% RSLogix 500 project P7 - Sensor Calibration.RSS, saved by version 8.30.00.16 %
PROJECT "P7"    % processor: Bul.1763 MicroLogix 1100 Series B %

PROGRAM FILES
  LAD 2 "MAIN"  3 rungs
  LAD 3 "IO"  3 rungs
  LAD 4 "SAMPLING"  4 rungs
  LAD 5 "CALIBRATE"  11 rungs

DATA FILES
  O0 OUTPUT  4 elements
  I1 INPUT  6 elements
  S2 STATUS  66 elements
  B3 BINARY  1 elements
  T4 TIMER  3 elements
  C5 COUNTER  1 elements
  R6 CONTROL  1 elements
  N7 INTEGER  8 elements
  F8 FLOAT  5 elements
  PD9 PD  1 elements

LADDER 2 "MAIN"
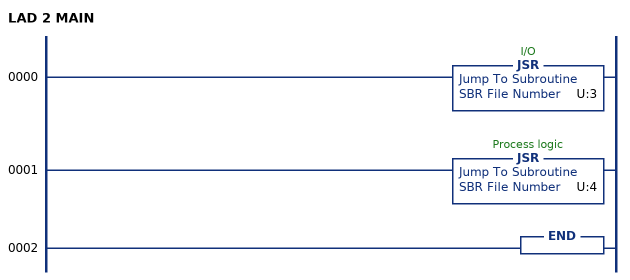
% Rung: 0 %
SOR JSR U:3 EOR
%   U:3  "I/O" %
% Rung: 1 %
SOR JSR U:4 EOR
%   U:4  "Process logic" %
% Rung: 2 %
SOR END EOR

LADDER 3 "IO"
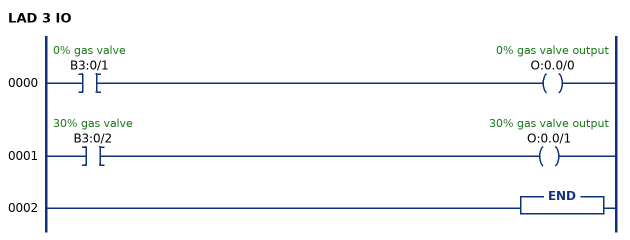
% Rung: 0 %
SOR XIC B3:0/1 OTE O:0.0/0 EOR
%   B3:0/1  "0% gas valve" %
%   O:0.0/0  "0% gas valve output" %
% Rung: 1 %
SOR XIC B3:0/2 OTE O:0.0/1 EOR
%   B3:0/2  "30% gas valve" %
%   O:0.0/1  "30% gas valve output" %
% Rung: 2 %
SOR END EOR

LADDER 4 "SAMPLING"
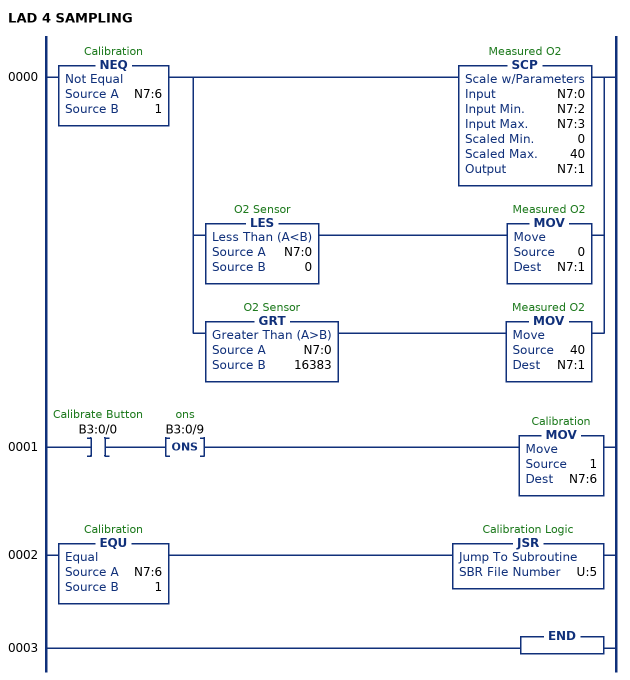
% Rung: 0 %
SOR NEQ N7:6 1 BST SCP N7:0 N7:2 N7:3 0 40 N7:1 NXB LES N7:0 0 MOV 0 N7:1 NXB GRT N7:0 16383 MOV 40 N7:1 BND EOR
%   N7:6  "Calibration" %
%   N7:0  "O2 Sensor" %
%   N7:2  "O2 min" %
%   N7:3  "O2 max" %
%   N7:1  "Measured O2" %
% Rung: 1 %
SOR XIC B3:0/0 ONS B3:0/9 MOV 1 N7:6 EOR
%   B3:0/0  "Calibrate Button" %
%   B3:0/9  "ons" %
%   N7:6  "Calibration" %
% Rung: 2 %
SOR EQU N7:6 1 JSR U:5 EOR
%   N7:6  "Calibration" %
%   U:5  "Calibration Logic" %
% Rung: 3 %
SOR END EOR

LADDER 5 "CALIBRATE"
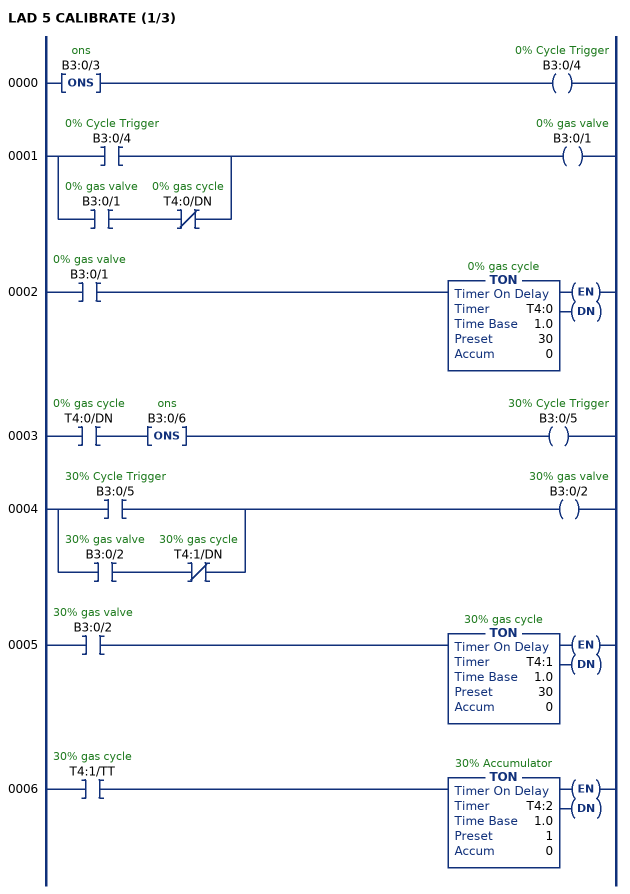
% Rung: 0 %
SOR ONS B3:0/3 OTE B3:0/4 EOR
%   B3:0/3  "ons" %
%   B3:0/4  "0% Cycle Trigger" %
% Rung: 1 %
SOR BST XIC B3:0/4 NXB XIC B3:0/1 XIO T4:0/DN BND OTE B3:0/1 EOR
%   B3:0/4  "0% Cycle Trigger" %
%   B3:0/1  "0% gas valve" %
%   T4:0  "0% gas cycle" %
% Rung: 2 %
SOR XIC B3:0/1 TON T4:0 1.0 30 0 EOR
%   B3:0/1  "0% gas valve" %
%   T4:0  "0% gas cycle" %
% Rung: 3 %
SOR XIC T4:0/DN ONS B3:0/6 OTE B3:0/5 EOR
%   T4:0  "0% gas cycle" %
%   B3:0/6  "ons" %
%   B3:0/5  "30% Cycle Trigger" %
% Rung: 4 %
SOR BST XIC B3:0/5 NXB XIC B3:0/2 XIO T4:1/DN BND OTE B3:0/2 EOR
%   B3:0/5  "30% Cycle Trigger" %
%   B3:0/2  "30% gas valve" %
%   T4:1  "30% gas cycle" %
% Rung: 5 %
SOR XIC B3:0/2 TON T4:1 1.0 30 0 EOR
%   B3:0/2  "30% gas valve" %
%   T4:1  "30% gas cycle" %
% Rung: 6 %
SOR XIC T4:1/TT TON T4:2 1.0 1 0 EOR
%   T4:1  "30% gas cycle" %
%   T4:2  "30% Accumulator" %

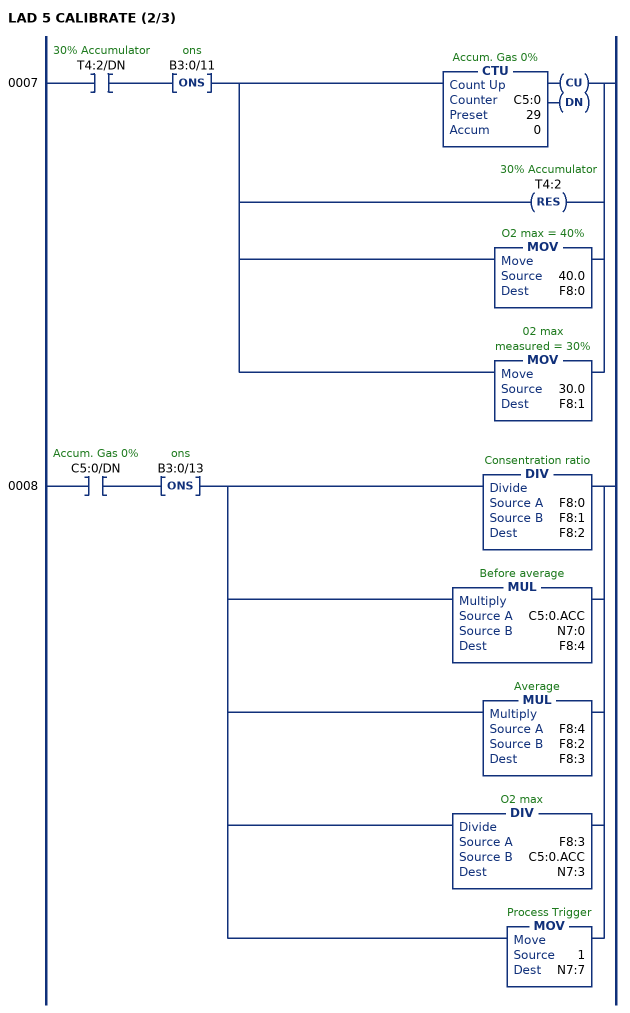
% Rung: 7 %
SOR XIC T4:2/DN ONS B3:0/11 BST CTU C5:0 29 0 NXB RES T4:2 NXB MOV 40.0 F8:0 NXB MOV 30.0 F8:1 BND EOR
%   T4:2/DN  "30% Accumulator" %
%   B3:0/11  "ons" %
%   C5:0  "Accum. Gas 0%" %
%   T4:2  "30% Accumulator" %
%   F8:0  "O2 max = 40%" %
%   F8:1  "02 max measured = 30%" %
% Rung: 8 %
SOR XIC C5:0/DN ONS B3:0/13 BST DIV F8:0 F8:1 F8:2 NXB MUL C5:0.ACC N7:0 F8:4 NXB MUL F8:4 F8:2 F8:3 NXB DIV F8:3 C5:0.ACC N7:3 NXB MOV 1 N7:7 BND EOR
%   C5:0  "Accum. Gas 0%" %
%   B3:0/13  "ons" %
%   F8:0  "O2 max = 40%" %
%   F8:1  "02 max measured = 30%" %
%   F8:2  "Consentration ratio" %
%   N7:0  "O2 Sensor" %
%   F8:4  "Before average" %
%   F8:3  "Average" %
%   N7:3  "O2 max" %
%   N7:7  "Process Trigger" %

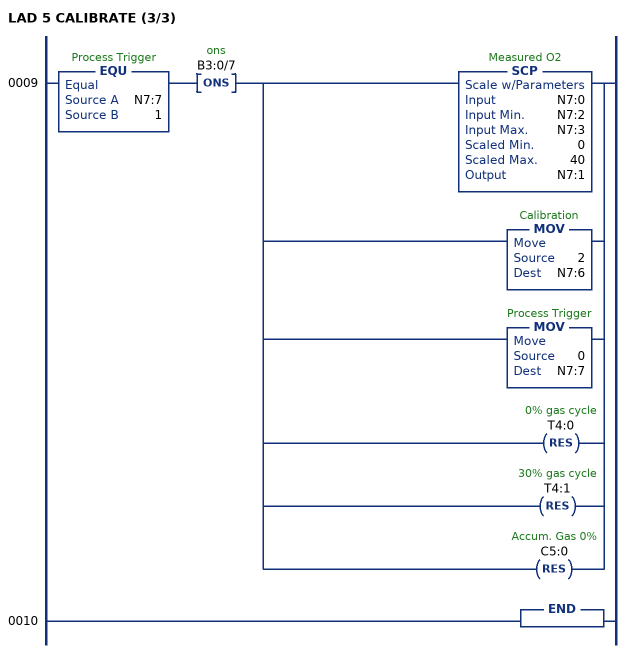
% Rung: 9 %
SOR EQU N7:7 1 ONS B3:0/7 BST SCP N7:0 N7:2 N7:3 0 40 N7:1 NXB MOV 2 N7:6 NXB MOV 0 N7:7 NXB RES T4:0 NXB RES T4:1 NXB RES C5:0 BND EOR
%   N7:7  "Process Trigger" %
%   B3:0/7  "ons" %
%   N7:0  "O2 Sensor" %
%   N7:2  "O2 min" %
%   N7:3  "O2 max" %
%   N7:1  "Measured O2" %
%   N7:6  "Calibration" %
%   T4:0  "0% gas cycle" %
%   T4:1  "30% gas cycle" %
%   C5:0  "Accum. Gas 0%" %
% Rung: 10 %
SOR END EOR

OTHER DOCUMENTED ADDRESSES
  B3:0/8  "ons"
  B3:0/10  "ons"
  B3:0/12  "Process trigger"
  N7:5  "Measured scaled"
  PD9:0  "0% gas cycle"

DATA TABLE (non-zero values as saved)
DATA T4
% .PRE .ACC %
% T4:0 % 30 0
% T4:1 % 30 0
% T4:2 % 1 0
DATA C5
% .PRE .ACC %
% C5:0 % 29 0
